{attribute 'linkalways'} 
{attribute 'no_explicit_call' := 'This FB is a CLASS and must be accessed using methods or properties'}
{attribute 'enable_dynamic_creation'}
FUNCTION_BLOCK PDFReport IMPLEMENTS I_ReportGenerator
VAR
	reportGenerateCommand : ReportGenerateCommand;
END_VAR

PROPERTY PUBLIC Busy : BOOL
GET
Busy := reportGenerateCommand.Busy;
END_GET
END_PROPERTY

METHOD PUBLIC CyclicCall
VAR_INPUT
END_VAR
IF reportGenerateCommand.Busy THEN
	reportGenerateCommand.CyclicCall();
END_IF
END_METHOD

PROPERTY PUBLIC Done : BOOL
GET
Done := reportGenerateCommand.Done;
END_GET
END_PROPERTY

PROPERTY PUBLIC Error : BOOL
GET
Error := reportGenerateCommand.Error;
END_GET
END_PROPERTY

PROPERTY PUBLIC ErrorId : UDINT
GET
ErrorId := reportGenerateCommand.ErrorId;
END_GET
END_PROPERTY

METHOD PUBLIC Generate
VAR_INPUT
	SourceData : ANY; // SourceData must be a Structure DUT
	TemplateName : T_MAXSTRING;
	FileName : T_MAXSTRING;
	FilePath : T_MAXSTRING;
END_VAR
reportGenerateCommand.Setup(
	SourceData := SourceData,
	TemplateName := TemplateName,
	FileName := FileName,
	FilePath := FilePath
);

reportGenerateCommand.Execute();
END_METHOD

END_FUNCTION_BLOCK

(* stored: Version 1.1.0.1, ProductVersion 3.1.4024.12
   POU PDFReport: Id {787c95bb-c8ef-408d-8304-be2e76ca35aa}, SpecialFunc None
   Property Busy: Id {572c63a6-3697-4981-8b18-dac8d61f36b8}
   Get Get: Id {1655fb7e-0d61-4aaf-9dc2-99be0833b8ab}
   Method CyclicCall: Id {cec7a61a-94b2-451a-80ac-4505bac16416}
   Property Done: Id {88367a11-3f10-4f05-9bab-7bd34a4217bc}
   Get Get: Id {7bf33be6-dc4f-4f67-8f3b-5d628f4983cd}
   Property Error: Id {6a7f5244-a9b9-4846-b9fc-7a542d0ad1a5}
   Get Get: Id {6434d8a4-9a87-44e9-9381-3938d5bf0e4d}
   Property ErrorId: Id {575e68ce-f570-4df3-a383-389888c2e549}
   Get Get: Id {f991e5f6-fc52-42ed-9487-85a357886abc}
   Method Generate: Id {4fa26abb-1031-47cf-9e78-31864f92535c} *)
